{attribute addProperty BoxType "KL9900-0059"}
{attribute addProperty Id "Key_1AT %I*BOOL000Key_2AT %I*BOOL000Key_3AT %I*BOOL000Key_4AT %I*BOOL000Key_5AT %I*BOOL000Key_6AT %I*BOOL000Key_7AT %I*BOOL000Key_8AT %I*BOOL000Key_9AT %I*BOOL000Key_10AT %I*BOOL000Key_11AT %I*BOOL000Key_12AT %I*BOOL000Key_13AT %I*BOOL000Key_14AT %I*BOOL000Key_15AT %I*BOOL000Key_16AT %I*BOOL000Key_17AT %I*BOOL000Key_18AT %I*BOOL000Key_19AT %I*BOOL000Key_20AT %I*BOOL000Key_21AT %I*BOOL000Key_22AT %I*BOOL000Key_23AT %I*BOOL000Key_24AT %I*BOOL000LED_1AT %Q*BOOL000LED_2AT %Q*BOOL000LED_3AT %Q*BOOL000LED_4AT %Q*BOOL000LED_5AT %Q*BOOL000LED_6AT %Q*BOOL000LED_7AT %Q*BOOL000LED_8AT %Q*BOOL000LED_9AT %Q*BOOL000LED_10AT %Q*BOOL000LED_11AT %Q*BOOL000LED_12AT %Q*BOOL000LED_13AT %Q*BOOL000LED_14AT %Q*BOOL000LED_15AT %Q*BOOL000LED_16AT %Q*BOOL000LED_17AT %Q*BOOL000LED_18AT %Q*BOOL000LED_19AT %Q*BOOL000LED_20AT %Q*BOOL000LED_21AT %Q*BOOL000LED_22AT %Q*BOOL000LED_23AT %Q*BOOL000LED_24AT %Q*BOOL000"}
{attribute addProperty CRC "1088792485"}
{attribute addProperty SizeInBites "0"}
{attribute addProperty SizeInBytes "0"}
TYPE Channel_40E5A7A5 :
STRUCT
	{attribute addProperty Name "Key_1"}
	Key_1 AT %I* : BOOL;
	{attribute addProperty Name "Key_2"}
	Key_2 AT %I* : BOOL;
	{attribute addProperty Name "Key_3"}
	Key_3 AT %I* : BOOL;
	{attribute addProperty Name "Key_4"}
	Key_4 AT %I* : BOOL;
	{attribute addProperty Name "Key_5"}
	Key_5 AT %I* : BOOL;
	{attribute addProperty Name "Key_6"}
	Key_6 AT %I* : BOOL;
	{attribute addProperty Name "Key_7"}
	Key_7 AT %I* : BOOL;
	{attribute addProperty Name "Key_8"}
	Key_8 AT %I* : BOOL;
	{attribute addProperty Name "Key_9"}
	Key_9 AT %I* : BOOL;
	{attribute addProperty Name "Key_10"}
	Key_10 AT %I* : BOOL;
	{attribute addProperty Name "Key_11"}
	Key_11 AT %I* : BOOL;
	{attribute addProperty Name "Key_12"}
	Key_12 AT %I* : BOOL;
	{attribute addProperty Name "Key_13"}
	Key_13 AT %I* : BOOL;
	{attribute addProperty Name "Key_14"}
	Key_14 AT %I* : BOOL;
	{attribute addProperty Name "Key_15"}
	Key_15 AT %I* : BOOL;
	{attribute addProperty Name "Key_16"}
	Key_16 AT %I* : BOOL;
	{attribute addProperty Name "Key_17"}
	Key_17 AT %I* : BOOL;
	{attribute addProperty Name "Key_18"}
	Key_18 AT %I* : BOOL;
	{attribute addProperty Name "Key_19"}
	Key_19 AT %I* : BOOL;
	{attribute addProperty Name "Key_20"}
	Key_20 AT %I* : BOOL;
	{attribute addProperty Name "Key_21"}
	Key_21 AT %I* : BOOL;
	{attribute addProperty Name "Key_22"}
	Key_22 AT %I* : BOOL;
	{attribute addProperty Name "Key_23"}
	Key_23 AT %I* : BOOL;
	{attribute addProperty Name "Key_24"}
	Key_24 AT %I* : BOOL;
	{attribute addProperty Name "LED_1"}
	LED_1 AT %Q* : BOOL;
	{attribute addProperty Name "LED_2"}
	LED_2 AT %Q* : BOOL;
	{attribute addProperty Name "LED_3"}
	LED_3 AT %Q* : BOOL;
	{attribute addProperty Name "LED_4"}
	LED_4 AT %Q* : BOOL;
	{attribute addProperty Name "LED_5"}
	LED_5 AT %Q* : BOOL;
	{attribute addProperty Name "LED_6"}
	LED_6 AT %Q* : BOOL;
	{attribute addProperty Name "LED_7"}
	LED_7 AT %Q* : BOOL;
	{attribute addProperty Name "LED_8"}
	LED_8 AT %Q* : BOOL;
	{attribute addProperty Name "LED_9"}
	LED_9 AT %Q* : BOOL;
	{attribute addProperty Name "LED_10"}
	LED_10 AT %Q* : BOOL;
	{attribute addProperty Name "LED_11"}
	LED_11 AT %Q* : BOOL;
	{attribute addProperty Name "LED_12"}
	LED_12 AT %Q* : BOOL;
	{attribute addProperty Name "LED_13"}
	LED_13 AT %Q* : BOOL;
	{attribute addProperty Name "LED_14"}
	LED_14 AT %Q* : BOOL;
	{attribute addProperty Name "LED_15"}
	LED_15 AT %Q* : BOOL;
	{attribute addProperty Name "LED_16"}
	LED_16 AT %Q* : BOOL;
	{attribute addProperty Name "LED_17"}
	LED_17 AT %Q* : BOOL;
	{attribute addProperty Name "LED_18"}
	LED_18 AT %Q* : BOOL;
	{attribute addProperty Name "LED_19"}
	LED_19 AT %Q* : BOOL;
	{attribute addProperty Name "LED_20"}
	LED_20 AT %Q* : BOOL;
	{attribute addProperty Name "LED_21"}
	LED_21 AT %Q* : BOOL;
	{attribute addProperty Name "LED_22"}
	LED_22 AT %Q* : BOOL;
	{attribute addProperty Name "LED_23"}
	LED_23 AT %Q* : BOOL;
	{attribute addProperty Name "LED_24"}
	LED_24 AT %Q* : BOOL;
END_STRUCT
END_TYPE

(* stored: Version 1.2.0.0, ProductVersion 3.1.4024.9
   DUT Channel_40E5A7A5: Id {789e8193-42d1-42b1-88e1-0e61d1f92c6d} *)
